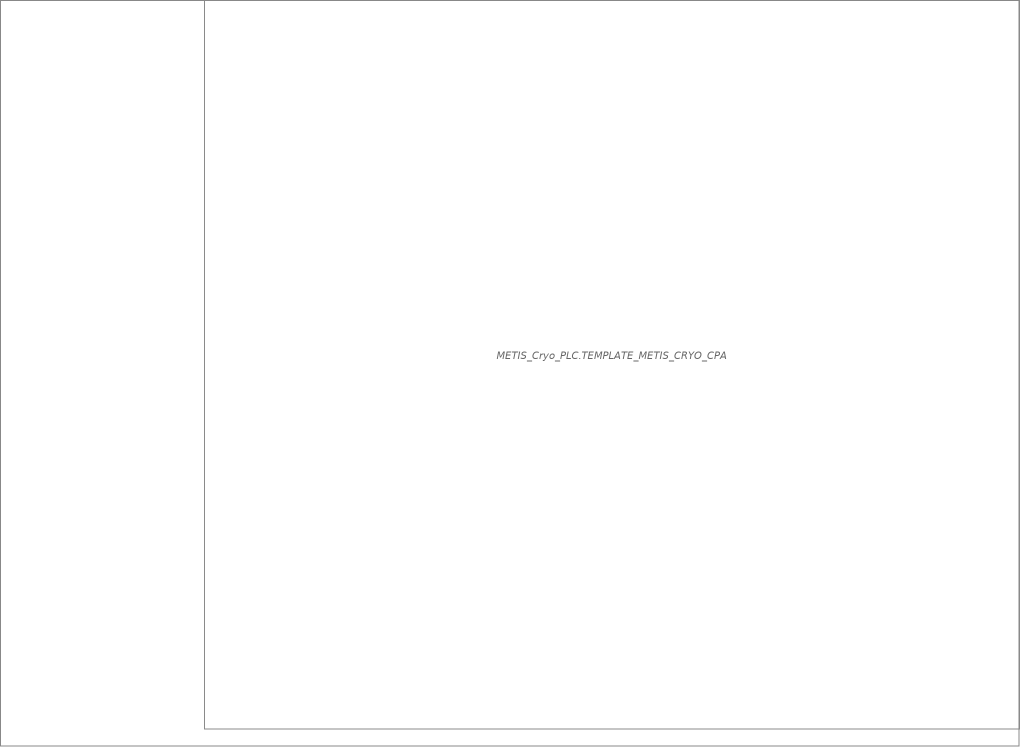
VISUALIZATION VISU_PTC_COOLER  // 1020x747
    Frame (204,-18 816x747)
        shows METIS_Cryo_PLC.TEMPLATE_METIS_CRYO_CPA(m_Instance := MAIN.nott_cryo_ctrl.cool_down.cooler, m_Cmd := MAIN.nott_cryo_ctrl.ctrl.cor_Cooler)
END_VISUALIZATION

(* stored: Version 1.1.0.1, ProductVersion 3.1.4026.18
   Visu VISU_PTC_COOLER: Id {c02f071a-e44a-49dd-8912-b45ade4f4f99} *)
